FUNCTION_BLOCK CROSSCOMM_PEER_239285CDFC5570564 (* Service Interface Function Block Type *)
  (* Standard: 61499-2 *)
  (* Version 0.0, 9/22/2017, bababen, nxtControl GmbH, template *)
  PACKAGE Main;
  (* Compiler Cpp nxtControl builtin 1.0 *)
  {SET_ATTRIBUTE(Runtime.FBType.ImplementingType, Runtime.System#DYNGEN_CROSSCOMM_PEER)}
  {SET_ATTRIBUTE(Configuration.GenericFBType.InterfaceParams, Runtime.System#<InterfaceList> <EventOutputs> <Event Name="CNF"> <With Var="PRetracked" /> <With Var="PExtended" /> </Event> </EventOutputs> <OutputVars> <VarDeclaration Name="PRetracked" Type="BOOL" /> <VarDeclaration Name="PExtended" Type="BOOL" /> </OutputVars> </InterfaceList>)}
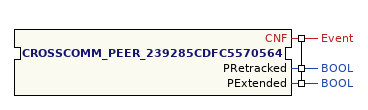
  EVENT_OUTPUT
    CNF WITH PRetracked, PExtended;
  END_EVENT
  VAR_OUTPUT
    PRetracked : BOOL;
    PExtended : BOOL;
  END_VAR
  EC_STATES
    START;
  END_STATES
END_FUNCTION_BLOCK
